// TIA Portal V20 export
// export: Created 2026-07-10T11:12:26.2872607Z, ExportSetting WithDefaults, DisplayName Totally Integrated Automation Portal, DisplayVersion V20, DisplayName TIA Portal Openness, DisplayVersion V20, DisplayName TIA Portal Version Control Interface, DisplayVersion V20, DisplayName STEP 7 Professional, DisplayVersion V20, DisplayName STEP 7 Safety, DisplayVersion V20, DisplayName WinCC Basic/Comfort/Advanced, DisplayVersion V20, DisplayName WinCC Unified, DisplayVersion V20
ORGANIZATION_BLOCK "DayOn"   // OB10, SCL, TimeOfDay
{ S7_Optimized_Access := 'TRUE' }
VERSION : 0.1
// stored: AutoNumber true, IsIECCheckEnabled false, SetENOAutomatically false
   VAR_INPUT
      CaughtUp : Bool;   // OB call is caught up because time was set forward
      SecondTime : Bool;   // OB call is started a second time because time was set backward
   END_VAR
BEGIN
   IF "MB".Table.HMI_CycleOn THEN
       "MB".Table.CycleDay := "MB".Table.CycleDay + 1;
       IF "MB".Table.CycleDay = "MB".Table.CycleStartDay[0] THEN
           "MB".Table.UsePID := TRUE;
       END_IF;
       IF "MB".Table.CycleDay = "MB".Table.CycleStartDay[4] THEN
           "MB".Table.UsePID := FALSE;
       END_IF;

       IF "MB".Table.CycleDay = "MB".Table.ChlorationCounter_SwitchDay AND "MB".Table.ChlorationCounter_SwitchOn THEN
           "MB".Table.Chloration_ChooseCounter := 1;
       END_IF;
   END_IF;
   "MB".Table.DayChangeFlag := TRUE;
   "MB".Table.WaterCounterIn_DailyCount := 0;
   "MB".Table.WaterCounterOut_DailyCount := 0;
   "MB".Table.Doser1_DailyPulses := 0;
   "MB".Table.Doser2_DailyPulses := 0;
END_ORGANIZATION_BLOCK
